// TwinCAT 3 PLC project RobotMainTask
// ProgramVersion: 3.1.4022.3
// libraries:
//   SysMem, * (System)
//   Tc2_MC2, * (Beckhoff Automation GmbH)
//   Tc2_SerialCom, * (Beckhoff Automation GmbH)
//   Tc2_Standard, * (Beckhoff Automation GmbH)
//   Tc2_System, * (Beckhoff Automation GmbH)
//   Tc2_TcpIp, * (Beckhoff Automation GmbH)
//   Tc3_Module, * (Beckhoff Automation GmbH)
// project tree:
//   / CommTask.TcTTO, MainTask.TcTTO
//   DUTs/ E_ExeCmd.TcDUT, E_MotorStatus.TcDUT, ST_AxisOut.TcDUT, ST_MoveObj.TcDUT, ST_PLCGroupSetAxis.TcDUT, ST_PLCSetAxis.TcDUT
//   GVLs/ GVL.TcGVL
//   POUs/ Comm.TcPOU, MAIN.TcPOU
//   POUs/Fuctions/ FB_ReadAxisStatus.TcPOU, FB_Robot.TcPOU, FB_SetAxisMotion.TcPOU, FB_RecvDataQue.TcPOU, FB_SendDataQue.TcPOU, FB_ServerWait.TcPOU
// real-time tasks:
//   TASK MainTask: cycle T#10ms, priority 8, ADS port 351
//   TASK CommTask: cycle T#20ms, priority 12, ADS port 352
// motion (NC):
//   TASK NC-Task 1 SAF: cycle T#2ms, priority 4, ADS port 501
//   TASK NC-Task 1 SVB: cycle T#10ms, priority 10, ADS port 511
//   AXIS Axis 1 (id 1)
//     OtherSettings: AllowMotionCmdToSlave=true
//     encoder EncType=19
//       EncPara: Offset=1210, MaxCount=#xffffffff
//     drive DrvType=16
//       DrvPara: MaxCount=#xffffffff, DriveControlDWord=#x00020000
//         Analog: ScaleFactorActTorque=0.1
//         TimeComp: TaskDelayCycles=1
//     controller CtrType=1
//       CtrPara: PriorControlFactor=1
//         Observer: BandWidth=20
//   AXIS Axis 2 (id 2)
//     OtherSettings: AllowMotionCmdToSlave=true
//     encoder EncType=19
//       EncPara: ScaleFactorDenominator=51.095748, Offset=1163.3371, Inverse=true, MaxCount=#xffffffff
//     drive DrvType=16
//       DrvPara: Inverse=true, MaxCount=#xffffffff, DriveControlDWord=#x00020000
//         Analog: ScaleFactorActTorque=0.1
//         TimeComp: TaskDelayCycles=1
//     controller CtrType=1
//       CtrPara: PriorControlFactor=1
//         Observer: BandWidth=20
//   AXIS Axis 3 (id 3)
//     OtherSettings: AllowMotionCmdToSlave=true
//     encoder EncType=19
//       EncPara: ScaleFactorDenominator=51.095748, Offset=318.369, Inverse=true, MaxCount=#xffffffff
//     drive DrvType=16
//       DrvPara: Inverse=true, MaxCount=#xffffffff, DriveControlDWord=#x00020000
//         Analog: ScaleFactorActTorque=0.1
//         TimeComp: TaskDelayCycles=1
//     controller CtrType=1
//       CtrPara: PriorControlFactor=1
//         Observer: BandWidth=20
//   AXIS Axis 4 (id 4)
//     OtherSettings: AllowMotionCmdToSlave=true
//     encoder EncType=19
//       EncPara: ScaleFactorDenominator=11.75751305, Offset=107.3187, Inverse=true, MaxCount=#xffffffff
//     drive DrvType=16
//       DrvPara: Inverse=true, MaxCount=#xffffffff, DriveControlDWord=#x00020000
//         Analog: ScaleFactorActTorque=0.1
//         TimeComp: TaskDelayCycles=1
//     controller CtrType=1
//       CtrPara: PriorControlFactor=1
//         Observer: BandWidth=20
//   AXIS Axis 5 (id 5)
//     OtherSettings: AllowMotionCmdToSlave=true
//     encoder EncType=19
//       EncPara: ScaleFactorDenominator=141.4214, Offset=4.8786, MaxCount=#xffffffff
//     drive DrvType=16
//       DrvPara: MaxCount=#xffffffff, DriveControlDWord=#x00020000
//         Analog: ScaleFactorActTorque=0.1
//         TimeComp: TaskDelayCycles=1
//     controller CtrType=1
//       CtrPara: PriorControlFactor=1
//         Observer: BandWidth=20
//   AXIS Axis 6 (id 6)
//     OtherSettings: AllowMotionCmdToSlave=true
//     encoder EncType=19
//       EncPara: ScaleFactorDenominator=5.22698, MaxCount=#xffffffff
//     drive DrvType=16
//       DrvPara: MaxCount=#xffffffff, DriveControlDWord=#x00020000
//         Analog: ScaleFactorActTorque=0.1
//         TimeComp: TaskDelayCycles=1
//     controller CtrType=1
//       CtrPara: PriorControlFactor=1
//         Observer: BandWidth=20
//   AXIS Axis 7 (id 7)
//     OtherSettings: AllowMotionCmdToSlave=true
//     encoder EncType=19
//       EncPara: ScaleFactorDenominator=5.25493, Offset=5, Inverse=true, MaxCount=#xffffffff
//     drive DrvType=16
//       DrvPara: Inverse=true, MaxCount=#xffffffff, DriveControlDWord=#x00020000
//         Analog: ScaleFactorActTorque=0.1
//         TimeComp: TaskDelayCycles=1
//     controller CtrType=1
//       CtrPara: PriorControlFactor=1
//         Observer: BandWidth=20
// I/O:
//   DEVICE Device 3 (EtherCAT), AmsNetId 192.168.1.240.4.1
//     Drive 1 (Elmo Drive) [Gold EtherCAT GCON Drive Rev:0x00010420]
//     Drive 2 (Elmo Drive) [Gold EtherCAT GCON Drive Rev:0x00010420]
//     Drive 3 (Elmo Drive) [Gold EtherCAT GCON Drive Rev:0x00010420]
//     Drive 4 (Elmo Drive) [Gold EtherCAT GCON Drive Rev:0x00010420]
//     Drive 5 (Elmo Drive) [Gold EtherCAT GCON Drive Rev:0x00010420]
//     Drive 6 (Elmo Drive) [Gold EtherCAT GCON Drive Rev:0x00010420]
//     Drive 7 (Elmo Drive) [Gold EtherCAT GCON Drive Rev:0x00010420]
//   DEVICE Device 2 (COM Port)
// variable links:
//   NC-Task 1 SAF/Axes/Axis 1 <-> Device 3 (EtherCAT)/Drive 1 (Elmo Drive)
//     Drive/Inputs/In/nDcOutputTime <-> InfoData/DcOutputShift
//     Drive/Inputs/In/nState1 <-> Inputs/Status word
//     Drive/Inputs/In/nState2 <-> Inputs/Status word @bit 8
//     Drive/Inputs/In/nState4 @bit 1 <-> WcState/InputToggle
//     Drive/Inputs/In/nState4 <-> WcState/WcState
//     Drive/Outputs/Out/nCtrl1 <-> Outputs/Control word
//     Drive/Outputs/Out/nCtrl2 <-> Outputs/Control word @bit 8
//     Drive/Outputs/Out/nDataOut1 <-> Outputs/Target Position
//     Enc/Inputs/In/nDataIn1 <-> Inputs/Position actual value
//     Enc/Inputs/In/nDcInputTime <-> InfoData/DcInputShift
//     Enc/Inputs/In/nState4 @bit 1 <-> WcState/InputToggle
//     Enc/Inputs/In/nState4 <-> WcState/WcState
//   NC-Task 1 SAF/Axes/Axis 2 <-> Device 3 (EtherCAT)/Drive 2 (Elmo Drive)
//     Drive/Inputs/In/nDcOutputTime <-> InfoData/DcOutputShift
//     Drive/Inputs/In/nState1 <-> Inputs/Status word
//     Drive/Inputs/In/nState2 <-> Inputs/Status word @bit 8
//     Drive/Inputs/In/nState4 @bit 1 <-> WcState/InputToggle
//     Drive/Inputs/In/nState4 <-> WcState/WcState
//     Drive/Outputs/Out/nCtrl1 <-> Outputs/Control word
//     Drive/Outputs/Out/nCtrl2 <-> Outputs/Control word @bit 8
//     Drive/Outputs/Out/nDataOut1 <-> Outputs/Target Position
//     Enc/Inputs/In/nDataIn1 <-> Inputs/Position actual value
//     Enc/Inputs/In/nDcInputTime <-> InfoData/DcInputShift
//     Enc/Inputs/In/nState4 @bit 1 <-> WcState/InputToggle
//     Enc/Inputs/In/nState4 <-> WcState/WcState
//   NC-Task 1 SAF/Axes/Axis 3 <-> Device 3 (EtherCAT)/Drive 3 (Elmo Drive)
//     Drive/Inputs/In/nDcOutputTime <-> InfoData/DcOutputShift
//     Drive/Inputs/In/nState1 <-> Inputs/Status word
//     Drive/Inputs/In/nState2 <-> Inputs/Status word @bit 8
//     Drive/Inputs/In/nState4 @bit 1 <-> WcState/InputToggle
//     Drive/Inputs/In/nState4 <-> WcState/WcState
//     Drive/Outputs/Out/nCtrl1 <-> Outputs/Control word
//     Drive/Outputs/Out/nCtrl2 <-> Outputs/Control word @bit 8
//     Drive/Outputs/Out/nDataOut1 <-> Outputs/Target Position
//     Enc/Inputs/In/nDataIn1 <-> Inputs/Position actual value
//     Enc/Inputs/In/nDcInputTime <-> InfoData/DcInputShift
//     Enc/Inputs/In/nState4 @bit 1 <-> WcState/InputToggle
//     Enc/Inputs/In/nState4 <-> WcState/WcState
//   NC-Task 1 SAF/Axes/Axis 4 <-> Device 3 (EtherCAT)/Drive 4 (Elmo Drive)
//     Drive/Inputs/In/nDcOutputTime <-> InfoData/DcOutputShift
//     Drive/Inputs/In/nState1 <-> Inputs/Status word
//     Drive/Inputs/In/nState2 <-> Inputs/Status word @bit 8
//     Drive/Inputs/In/nState4 @bit 1 <-> WcState/InputToggle
//     Drive/Inputs/In/nState4 <-> WcState/WcState
//     Drive/Outputs/Out/nCtrl1 <-> Outputs/Control word
//     Drive/Outputs/Out/nCtrl2 <-> Outputs/Control word @bit 8
//     Drive/Outputs/Out/nDataOut1 <-> Outputs/Target Position
//     Enc/Inputs/In/nDataIn1 <-> Inputs/Position actual value
//     Enc/Inputs/In/nDcInputTime <-> InfoData/DcInputShift
//     Enc/Inputs/In/nState4 @bit 1 <-> WcState/InputToggle
//     Enc/Inputs/In/nState4 <-> WcState/WcState
//   NC-Task 1 SAF/Axes/Axis 5 <-> Device 3 (EtherCAT)/Drive 5 (Elmo Drive)
//     Drive/Inputs/In/nDcOutputTime <-> InfoData/DcOutputShift
//     Drive/Inputs/In/nState1 <-> Inputs/Status word
//     Drive/Inputs/In/nState2 <-> Inputs/Status word @bit 8
//     Drive/Inputs/In/nState4 @bit 1 <-> WcState/InputToggle
//     Drive/Inputs/In/nState4 <-> WcState/WcState
//     Drive/Outputs/Out/nCtrl1 <-> Outputs/Control word
//     Drive/Outputs/Out/nCtrl2 <-> Outputs/Control word @bit 8
//     Drive/Outputs/Out/nDataOut1 <-> Outputs/Target Position
//     Enc/Inputs/In/nDataIn1 <-> Inputs/Position actual value
//     Enc/Inputs/In/nDcInputTime <-> InfoData/DcInputShift
//     Enc/Inputs/In/nState4 @bit 1 <-> WcState/InputToggle
//     Enc/Inputs/In/nState4 <-> WcState/WcState
//   NC-Task 1 SAF/Axes/Axis 6 <-> Device 3 (EtherCAT)/Drive 6 (Elmo Drive)
//     Drive/Inputs/In/nDataIn3[0] <-> Inputs_1/Torque actual value
//     Drive/Inputs/In/nDcOutputTime <-> InfoData/DcOutputShift
//     Drive/Inputs/In/nState1 <-> Inputs/Status word
//     Drive/Inputs/In/nState2 <-> Inputs/Status word @bit 8
//     Drive/Inputs/In/nState4 @bit 1 <-> WcState/InputToggle
//     Drive/Inputs/In/nState4 <-> WcState/WcState
//     Drive/Outputs/Out/nCtrl1 <-> Outputs/Control word
//     Drive/Outputs/Out/nCtrl2 <-> Outputs/Control word @bit 8
//     Drive/Outputs/Out/nDataOut1 <-> Outputs/Target Position
//     Enc/Inputs/In/nDataIn1 <-> Inputs/Position actual value
//     Enc/Inputs/In/nDcInputTime <-> InfoData/DcInputShift
//     Enc/Inputs/In/nState4 @bit 1 <-> WcState/InputToggle
//     Enc/Inputs/In/nState4 <-> WcState/WcState
//   NC-Task 1 SAF/Axes/Axis 7 <-> Device 3 (EtherCAT)/Drive 7 (Elmo Drive)
//     Drive/Inputs/In/nDcOutputTime <-> InfoData/DcOutputShift
//     Drive/Inputs/In/nState1 <-> Inputs/Status word
//     Drive/Inputs/In/nState2 <-> Inputs/Status word @bit 8
//     Drive/Inputs/In/nState4 @bit 1 <-> WcState/InputToggle
//     Drive/Inputs/In/nState4 <-> WcState/WcState
//     Drive/Outputs/Out/nCtrl1 <-> Outputs/Control word
//     Drive/Outputs/Out/nCtrl2 <-> Outputs/Control word @bit 8
//     Drive/Outputs/Out/nDataOut1 <-> Outputs/Target Position
//     Enc/Inputs/In/nDataIn1 <-> Inputs/Position actual value
//     Enc/Inputs/In/nDcInputTime <-> InfoData/DcInputShift
//     Enc/Inputs/In/nState4 @bit 1 <-> WcState/InputToggle
//     Enc/Inputs/In/nState4 <-> WcState/WcState
//   RobotMainTask/RobotMainTask Instance <-> Device 3 (EtherCAT)/Drive 6 (Elmo Drive)
//     CommTask Inputs/GVL.axisTorque <-> Inputs_1/Torque actual value
//   RobotMainTask/RobotMainTask Instance <-> NC-Task 1 SAF/Axes/Axis 1
//     MainTask Inputs/GVL.TestMotor[0].NcToPlc <-> Outputs/ToPlc
//     MainTask Outputs/GVL.TestMotor[0].PlcToNc <-> Inputs/FromPlc
//   RobotMainTask/RobotMainTask Instance <-> NC-Task 1 SAF/Axes/Axis 2
//     MainTask Inputs/GVL.TestMotor[1].NcToPlc <-> Outputs/ToPlc
//     MainTask Outputs/GVL.TestMotor[1].PlcToNc <-> Inputs/FromPlc
//   RobotMainTask/RobotMainTask Instance <-> NC-Task 1 SAF/Axes/Axis 3
//     MainTask Inputs/GVL.TestMotor[2].NcToPlc <-> Outputs/ToPlc
//     MainTask Outputs/GVL.TestMotor[2].PlcToNc <-> Inputs/FromPlc
//   RobotMainTask/RobotMainTask Instance <-> NC-Task 1 SAF/Axes/Axis 4
//     MainTask Inputs/GVL.TestMotor[3].NcToPlc <-> Outputs/ToPlc
//     MainTask Outputs/GVL.TestMotor[3].PlcToNc <-> Inputs/FromPlc
//   RobotMainTask/RobotMainTask Instance <-> NC-Task 1 SAF/Axes/Axis 5
//     MainTask Inputs/GVL.TestMotor[4].NcToPlc <-> Outputs/ToPlc
//     MainTask Outputs/GVL.TestMotor[4].PlcToNc <-> Inputs/FromPlc
//   RobotMainTask/RobotMainTask Instance <-> NC-Task 1 SAF/Axes/Axis 6
//     MainTask Inputs/GVL.TestMotor[5].NcToPlc <-> Outputs/ToPlc
//     MainTask Outputs/GVL.TestMotor[5].PlcToNc <-> Inputs/FromPlc
//   RobotMainTask/RobotMainTask Instance <-> NC-Task 1 SAF/Axes/Axis 7
//     MainTask Inputs/GVL.TestMotor[6].NcToPlc <-> Outputs/ToPlc
//     MainTask Outputs/GVL.TestMotor[6].PlcToNc <-> Inputs/FromPlc

CONFIGURATION RobotMainTask
    RESOURCE PLC ON TwinCAT3
        TASK CommTask(INTERVAL := T#20ms, PRIORITY := 12);
        TASK MainTask(INTERVAL := T#10ms, PRIORITY := 8);
        PROGRAM Comm WITH CommTask : Comm;
        PROGRAM MAIN WITH MainTask : MAIN;
    END_RESOURCE
END_CONFIGURATION

// ---- DUTs/E_ExeCmd.TcDUT
{attribute 'qualified_only'}
{attribute 'strict'}
TYPE E_ExeCmd :
(
		E_PowerOff,
		E_PowerOn,    //E_Enable
		E_MoveAbs,
		E_MoveConAbs,
		E_MoveRelative,
		E_MoveVelocity,
		E_Halt,
		E_Stop,
		E_Reset,
		E_Home
);
END_TYPE

// ---- DUTs/E_MotorStatus.TcDUT
{attribute 'qualified_only'}
{attribute 'strict'}
TYPE E_MotorStatus :
(
	MOTORSTATUS_DISABLED,       	//*****NEW	if the MC_Power.Enable is FALSE that motor will be disable, from any MOTORSTATUS
	MOTORSTATUS_Standstill,		//is the enable status, can response any Cmd
	MOTORSTATUS_ERRORSTOP,		//NEW
	MOTORSTATUS_HOMING,			//NEW
	MOTORSTATUS_STOPPING,		//NEW
	MOTORSTATUS_DISCRETEMOTION,		//NEW
	MOTORSTATUS_CONTINUOUSMOTION,	//NEW
	MOTORSTATUS_SYNMOTION		//Advance
);
END_TYPE

// ---- DUTs/ST_AxisOut.TcDUT
TYPE ST_AxisOut :
STRUCT


	eStatus   : E_MotorStatus;
	
	Response 	: STRING;
	ENABLE     : BOOL;
	ServoDone  : BOOL;
	ServoBusy  : BOOL;
	ServoError : BOOL;
	ServoErrorID : UDINT;	
//get these variable from the READSTATUS().NcToPlc;	
//	ErrorCode:UDINT;//NC轴错误代码
//	AxisState:UDINT;//NC轴状态
//	HomingState:UDINT;//NC轴回原位状态
//	AxisId:UDINT;//NC轴的编码
	ActPos:LREAL;//NC轴的实际位置
	ActVelo:LREAL;//NC轴的实际速度
	ActAcc:LREAL;//NC轴的实际加速度
	ActTorque:LREAL;//NC轴的实际转矩
	SetPos:LREAL;//NC轴的设定位置
	SetVelo:LREAL;//NC轴的设定速度
	SetAcc:LREAL;//NC轴的设定加速度
	SetTorque:LREAL;//NC轴的设定转矩
//	TargetPos:LREAL;//NC轴的目标位置
	PosDiff:LREAL;//位置误差	

END_STRUCT
END_TYPE

// ---- DUTs/ST_MoveObj.TcDUT
TYPE ST_MoveObj :
STRUCT
	
	Dir			: INT;	
	Position 		: LREAL;
	Distance 		: LREAL;
	Velocity 		: LREAL;
	EndVelocity 	: LREAL;
	Torque		: LREAL;

END_STRUCT
END_TYPE

// ---- DUTs/ST_PLCGroupSetAxis.TcDUT
TYPE ST_PLCGroupSetAxis :
STRUCT
	
	st_EachSetAxis : ARRAY [0..19] OF ST_PLCSetAxis;

END_STRUCT
END_TYPE

// ---- DUTs/ST_PLCSetAxis.TcDUT
TYPE ST_PLCSetAxis :
STRUCT
	
	Num  				: UINT;

	E_ExecuteCmd		: E_ExeCmd;
	ST_MoveObject		: ST_MoveObj;
		
END_STRUCT
END_TYPE

// ---- GVLs/GVL.TcGVL

{attribute 'qualified_only'}
VAR_GLOBAL
END_VAR
VAR_GLOBAL CONSTANT
	Reconnect_time 	: TIME := T#1S;
	ListenTime		: TIME := T#1S;
	AcceptTime		: TIME := T#1S;
	RecvTime 		: TIME := T#1S;	
	MaxDataLen		: UDINT := 3500;
	QueLen			: USINT := 4;
END_VAR
VAR_GLOBAL
	InitPar 		: st_InitParameter;
	// put new to tail and get data from heand  circularly
	fbRecvDataQue   : FB_RecvDataQue;
	fbSendDataQue 	: FB_SendDataQue;
	
	//NEW
	TestMotor : ARRAY [0..19] OF AXIS_REF;
END_VAR

// ---- POUs/Comm.TcPOU
PROGRAM Comm
VAR
	fbWaitConnect 	: FB_ServerWait;
	fbRecv			: FB_SocketReceive 	:= (sSrvNetId := '');
	fbSend			: FB_SocketSend 	:= (sSrvNetId := '');
	fbClose			: FB_SocketClose 	:= (sSrvNetID := '');	
	fbCloseAll		: FB_SocketCloseAll := (sSrvNetID := '');
	
	hSocket 		: T_HSOCKET;
	RecvLen 		: UDINT := 0;
	SendLen			: UDINT	:= 0;

	bNewRecv 		: BOOL;	
	bNewSend 		: BOOL;	
	bConnect 		: BOOL;
	nErrID 			: UDINT;
	step 			: UDINT;

	RecvBuff 		: ARRAY[1..GVL.MaxDataLen] OF BYTE;
	//SendBuff 		: ARRAY[1..GVL.DataLen] OF BYTE;
	SendBuff 		: ARRAY[1..GVL.MaxDataLen] OF BYTE;	
	DataRecv 		: ARRAY[1..GVL.MaxDataLen] OF BYTE;
	DataSend		: ARRAY[1..GVL.MaxDataLen] OF BYTE;
END_VAR

VAR(*For Test*)
	GetTime			: GETCPUACCOUNT;
	time_start		: UDINT;
	time_end 		: UDINT;
	time_cost 		: REAL;
END_VAR

CASE step OF
	0:(*prepare*)
		bConnect := FALSE;
		fbCloseAll(bExecute:= FALSE);
		fbCloseAll(bExecute:= TRUE);
		step := 1;
	1:(*Preparing*)
		fbCloseAll(bExecute:= FALSE);
		IF NOT fbCloseALL.bBusy THEN
			IF NOT fbCloseALL.bError THEN
				step := 5;
			ELSE 
				nErrID := fbCloseALL.nErrId;
				step := 0;
			END_IF
		END_IF
	5:(*wait for connect*)
		bConnect := FALSE;
		fbWaitConnect(bEnable := TRUE);
		nErrID := fbWaitConnect.nErrID;
		IF NOT fbWaitConnect.bBusy THEN
			IF NOT fbWaitConnect.bError THEN
				hSocket := fbWaitConnect.hSocket;
				step := 9;			
			ELSE
				nErrID := fbWaitConnect.nErrID;
			END_IF
		END_IF
		
	9:(*prepare to recieve data*)
		IF(GVL.InitPar.RecvSize <> 0) THEN
			fbRecv(bExecute := FALSE);
			bNewRecv := TRUE;
			bConnect := TRUE;
			RecvLen := GVL.InitPar.RecvSize;
			SendLen := GVL.InitPar.SendSize;
			step := 10;
			GVL.fbRecvDataQue.Reset();//Init recieve data queue
			GVL.fbSendDataQue.Reset();
		END_IF
		
		
	10:(*Receive and send phase I*)
		//*Start to recieve data
		fbRecv(hSocket := hSocket, cbLen := RecvLen, pDest := ADR(RecvBuff), bExecute := TRUE, tTimeout := GVL.RecvTime);
		//*prepare data to send
		fbSend(bExecute := FALSE);
		//Get SendData
		IF NOT fbSend.bBusy THEN
			IF NOT fbSend.bError THEN
				GVL.fbSendDataQue.GetFromQue(ADR(DataSend));
				step := 15;
			ELSE
				nErrID := fbSend.nErrId;
				step := 100;
			END_IF
		END_IF		
		step := 15;
	15: (*Receive and send phase II*)
		//deal with recieve data
		fbRecv(bExecute := FALSE);
		IF NOT fbRecv.bBusy THEN
			IF NOT fbRecv.bError THEN
				ACT_RecvData();
				IF bNewRecv THEN (*put databuff into recieve queque*)
					GVL.fbRecvDataQue.PutToQue(ADR(DataRecv));	
					memset(ADR(DataRecv),0, GVL.InitPar.RecvSize);		
				END_IF
				step := 10;			
			ELSE
				nErrID := fbRecv.nErrId;
				step := 100;	
			END_IF
		END_IF
		//SendData
		GVL.fbSendDataQue.GetFromQue(ADR(DataSend));
		
		IF GVL.fbSendDataQue.bGetData THEN
			fbSend(hSocket := hSocket,cbLen :=SendLen, pSrc := ADR(DataSend),bExecute := TRUE,tTimeout := gvl.RecvTime);
		END_IF
	100:(*deal with error*)
		bConnect := FALSE;
		fbClose(bExecute := FALSE);
		fbClose(hSocket := hSocket, bExecute := TRUE);
		step := 102;
	102: 
		bConnect := FALSE;
		fbClose(bExecute := FALSE);
		IF NOT fbClose.bBusy THEN
			IF NOT fbClose.bError THEN
				step:= 5;
			ELSE 
				step := 0;
			END_IF
		END_IF			
END_CASE

ACTION ACT_PreSend:

END_ACTION

ACTION ACT_RecvData:
(*Recieve data, every group of data has length of Datalen*)
IF bNewRecv THEN
	IF fbRecv.nRecBytes < GVL.InitPar.RecvSize THEN
		bNewRecv := FALSE;
		memcpy(ADR(DataRecv),ADR(RecvBuff),fbRecv.nRecBytes);
		RecvLen := GVL.InitPar.RecvSize - fbRecv.nRecBytes;
	ELSE
		memcpy(ADR(DataRecv),ADR(RecvBuff),GVL.InitPar.RecvSize);
		bNewRecv := TRUE;
	END_IF
ELSE
	IF fbRecv.nRecBytes < RecvLen THEN
		memcpy(ADR(DataRecv)+ GVL.InitPar.RecvSize - RecvLen, ADR(RecvBuff),fbRecv.nRecBytes);
		RecvLen := RecvLen - fbRecv.nRecBytes;
	ELSE		
		memcpy(ADR(DataRecv)+ GVL.InitPar.RecvSize - RecvLen, ADR(RecvBuff),RecvLen);
		bNewRecv := TRUE;
		RecvLen :=GVL.InitPar.RecvSize;
	END_IF					
END_IF
END_ACTION

END_PROGRAM

// ---- POUs/Fuctions/FB_ServerWait.TcPOU
FUNCTION_BLOCK FB_ServerWait
(*Listioning and accecpt connect for remote*)
VAR_INPUT
	bEnable : BOOL;
	sLocalHost : STRING(15) := '192.168.1.245';//'192.168.1.245';'192.168.137.74'
	nLocalPort : UINT := 4999;

END_VAR
VAR_OUTPUT
	hSocket : T_HSOCKET;
	bBusy: BOOL;
	bError: BOOL;
	nErrID : UDINT;
END_VAR
VAR
	fblisten :FB_SocketListen := (sSrvNetID := '');	
	fbAccept : FB_SocketAccept;
	fbClose : FB_SocketClose;
	fbReconncetTon: TON:=(PT := GVL.Reconnect_time);
	fbAcceptTon: TON:=(PT := GVL.AcceptTime);
		
	hListener : T_HSOCKET;	
	
	bListening : BOOL;
	bAccepting : BOOL;
	
	step : UINT := 0;
	
END_VAR

CASE step OF
	0:(*Init*)
		IF bEnable THEN
			fbReconncetTon(IN := FALSE);
			fblisten(bExecute := FALSE);
			step := 10;
			bBusy:= TRUE;
			nErrID := 0;
			bError := FALSE;
		END_IF
	10:(*Start listenin*)
		fbReconncetTon(IN := TRUE, PT := GVL.Reconnect_time);
		IF fbReconncetTon.Q THEN
			fblisten(sLocalHost := sLocalHost,
			nLocalPort := nLocalPort,
			bExecute := TRUE,
			tTimeout := GVL.ListenTime);
			step := 15;	
		END_IF
						
	15:(*Listening*)
		fbListen(bExecute := FALSE);
		bListening := TRUE;
		IF NOT fbListen.bBusy THEN
			IF NOT fbListen.bError THEN
				hListener := fbListen.hListener; 
				
				step := 20;
				(*prepare for accept*)
				fbAcceptTon(IN:=FALSE);
				fbAccept(bExecute := FALSE);
			ELSE
				bError := TRUE;				
				nErrID := fbListen.nErrId;
				step := 100;
			END_IF
		END_IF
	20:(*start to accept*)	
		bListening := FALSE;
		fbAcceptTon(IN := TRUE,PT := GVL.AcceptTime);
		IF fbAcceptTon.Q THEN
			fbAcceptTon(IN :=FALSE);
			fbAccept(hListener := hListener, bExecute := TRUE);
			step := 25;
		END_IF
	25: (* Accepting*)
		fbAccept(bExecute := FALSE);
		bAccepting := TRUE;
		IF NOT fbAccept.bBusy THEN
			IF NOT fbAccept.bError THEN
				(*check if there is connection be accepted*)
				IF fbAccept.bAccepted THEN
					hSocket := fbAccept.hSocket;
					bBusy := FALSE;
					step := 40;
				ELSE
					step := 20;
				END_IF	
							
			ELSE
				bError := TRUE;
				nErrID := fbAccept.nErrId;
				step := 100;	
			END_IF
		END_IF
		
	40:(*wait for new connect*)
		bBusy := TRUE;
		step:= 20;
	100:(*deal with error*)
		step := 0;
		
		
END_CASE

END_FUNCTION_BLOCK

// ---- POUs/MAIN.TcPOU

 PROGRAM MAIN
VAR{varable needed}
	robot				: FB_Robot;
	fbReadAxisStatus 	: FB_ReadAxisStatus;
	fbMCMotion 			: ARRAY[0..19] OF FB_SetAxisMotion;
	
	MC_ActStatus		: st_AxisGroupRead; 		 //**OUT**give the data to thr Upper
	MC_SetCommd			: st_AxisGroupSet;			 //**IN** get the data from the Upper and set the Axis 
	CtlComd		: RecvBuff;		(*Commd to MC*)
	Status		: SendBuff;		(*MC_State*)
	
	
	ErrID		: UDINT := 0;	
	step		: INT := 0;
	{time cost of every cycle}
	CycleTime	: LREAL := 0;
	CycleTime_Max: LREAL := 0;	
END_VAR

VAR{varable FOR test}
	i :UDINT := 0;
	j :UDINT := 0;
	w :UDINT := 0;
	vel : LREAL;
	nCounter: BYTE := 0;
	nCounter1: BYTE := 0;
	GetTime:GETCPUACCOUNT;
	time_start: UDINT;
	time_end:UDINT;
	labelOld:DINT := 0;
	labelNew:DINT := 0;
	count: UDINT := 0;
	count11 : UDINT := 0;
	delay : TON;
	
	test : LREAL := 0;
	test1 : LREAL := 0;
END_VAR

CASE step OF
	0: {prepare varable before start robot}	
		step := 5;
	5:	{NC init before robot start}	
		GroupInitAxis(); 	
		step := 10;
	10:{Init robot}
		ErrID := robot.InitRobot(ADR(GVL.InitPar));
	 	IF (0 = ErrID )THEN
		 	step := 15;
		ELSE
			step := 0;
		END_IF
	15:
		GetTime(cpuAccountDW=>time_start);
	 	
		GVL.fbRecvDataQue.GetfromQue(ADR(CtlComd));
		GroupReadAxis();

		robot.RunRobot(pMC_Inputs := ADR(MC_ActStatus), pMC_Outputs := ADR(MC_SetCommd),
								pCtlComd	:= ADR(CtlComd) , pRobotStatus := ADR(Status));
														
		GroupSetAxis();
		GVL.fbSendDataQue.PutToQue(ADR(Status));
		
		GetTime(cpuAccountDW=>time_end);
		CycleTime := (time_end- time_start)/10000.0;
		CycleTime_Max:= MAX(CycleTime,CycleTime_Max);
	 	
	20: 
		robot.StopRobot();
		step:= 0;
END_CASE;

ACTION GroupInitAxis:
i := 0;
END_ACTION

ACTION GroupReadAxis:
FOR i:= 0 TO 7 DO //MC_ActStatus.Number
	fbReadAxisStatus(AxisRef := GVL.TestMotor[i], AxisStatus => MC_ActStatus.AxisGoup[i]);	
END_FOR
END_ACTION

ACTION GroupSetAxis:
FOR i:= 0 TO 7 DO //MC_ActStatus.Number
	fbMCMotion[i](axis := GVL.TestMotor[i], SetCmd := MC_SetCommd.AxisGroup[i], ActStatus := MC_ActStatus.AxisGoup[i]);
END_FOR
//fbMCMotion(axis := GVL.TestMotor[0], SetCmd := MC_SetCommd.AxisGroup[0], ActStatus := MC_ActStatus.AxisGoup[0]);
END_ACTION

END_PROGRAM

// ---- POUs/Fuctions/FB_Robot.TcPOU
FUNCTION_BLOCK FB_Robot
VAR_INPUT
END_VAR
VAR_OUTPUT
END_VAR
VAR
	{attribute 'TcInitSymbol'}
	oidInstance : OTCID;
	ipRobot : IRobot;
	hrInit : HRESULT;
END_VAR

METHOD FB_exit : BOOL
VAR_INPUT
	bInCopyCode : BOOL; // if TRUE, the exit method is called for exiting an instance that is copied afterwards (online change).
END_VAR
IF NOT bInCopyCode THEN
	FW_SafeRelease(ADR(ipRobot));
END_IF
END_METHOD

METHOD FB_init : BOOL
VAR_INPUT
	bInitRetains : BOOL; // if TRUE, the retain variables are initialized (warm start / cold start)
	bInCopyCode : BOOL;  // if TRUE, the instance afterwards gets moved into the copy code (online change)
END_VAR
IF NOT bInCopyCode THEN
	IF ipRobot = 0 THEN
		hrInit := FW_objMgr_GetObjectInstance(oid := oidInstance, iid:= TC_GLOBAL_IID_LIST.IID_IRobot,pipUnk := ADR(ipRobot)); 
	END_IF
END_IF
END_METHOD

{attribute 'c++_compatible'}
{attribute 'minimal_input_size' := '4'}
{attribute 'pack_mode' := '4'}
{warning 'add method implementation'}
METHOD InitRobot : UDINT
VAR_INPUT
	pInitPar	: POINTER TO st_InitParameter;
END_VAR
IF (ipRobot <> 0) THEN
	InitRobot := ipRobot.InitRobot(pInitPar);
END_IF
END_METHOD


{attribute 'c++_compatible'}
{attribute 'minimal_input_size' := '4'}
{attribute 'pack_mode' := '4'}


METHOD RunRobot : UDINT
VAR_INPUT
	pMC_Inputs	: POINTER TO st_AxisGroupRead;
	pMC_Outputs	: POINTER TO st_AxisGroupSet;
	pCtlComd	: POINTER TO Recvbuff;
	pRobotStatus	: POINTER TO Sendbuff;
END_VAR
IF (ipRobot <> 0) THEN
	RunRobot := ipRobot.RunRobot(pMC_Inputs, pMC_Outputs, pCtlComd, pRobotStatus);
END_IF
END_METHOD

{attribute 'c++_compatible'}
{attribute 'minimal_input_size' := '4'}
{attribute 'pack_mode' := '4'}
{warning 'add method implementation'}
METHOD StopRobot : HRESULT
IF (ipRobot <> 0) THEN
	StopRobot := ipRobot.StopRobot();
END_IF
END_METHOD

END_FUNCTION_BLOCK

// ---- POUs/Fuctions/FB_ReadAxisStatus.TcPOU
FUNCTION_BLOCK FB_ReadAxisStatus
VAR_IN_OUT

AxisRef : AXIS_REF;

END_VAR

VAR_OUTPUT

AxisStatus : st_ReadAxis;

END_VAR
VAR	
END_VAR

AxisRef.ReadStatus();  
AxisStatus.Position			:= AxisRef.NcToPlc.ActPos;
AxisStatus.Velocity			:= AxisRef.NcToPlc.ActVelo;
AxisStatus.Acceleration		:= AxisRef.NcToPlc.ActAcc;
AxisStatus.Torque		    := AxisRef.NcToPlc.ActTorque;
//AxisStatus.Current			:= AxisRef.NcToPlc.ActTorque;
AxisStatus.ErrorID			:= AxisRef.NcToPlc.ErrorCode;

IF AxisRef.Status.ErrorStop THEN
	AxisStatus.eState := eAxis_ERRORSTOP;
ELSIF AxisRef.Status.Disabled THEN
	AxisStatus.eState := eAxis_DISABLED;
ELSIF AxisRef.Status.StandStill THEN
	AxisStatus.eState := eAxis_STANDSTILL;
ELSIF AxisRef.Status.Homing THEN
	AxisStatus.eState := eAxis_HOMING;
ELSIF AxisRef.Status.Stopping THEN
	AxisStatus.eState := eAxis_STOPPING;
ELSIF AxisRef.Status.DiscreteMotion THEN
	AxisStatus.eState := eAxis_DISCRETEMOTION;
ELSIF AxisRef.Status.ContinuousMotion THEN
	AxisStatus.eState := eAxis_CONTINOUSMOTION;
ELSIF AxisRef.Status.SynchronizedMotion THEN
	AxisStatus.eState := eAxis_SYNCHRONIZEDMOTION;
ELSE
	AxisStatus.eState := eAxis_UNDEFINED;
END_IF

END_FUNCTION_BLOCK

// ---- POUs/Fuctions/FB_SetAxisMotion.TcPOU
FUNCTION_BLOCK FB_SetAxisMotion
VAR_IN_OUT
		axis : AXIS_REF;   			// the input axis
END_VAR
VAR_INPUT
	SetCmd : st_SetAxis;	
	ActStatus: st_ReadAxis;
END_VAR
VAR		
	fbMC_Stop:			MC_Stop;		
	fbMC_Home:			MC_Home;		
	fbMC_Halt:			MC_Halt;
	fbMC_Power:			MC_Power;
	fbMC_Reset:			MC_Reset;
	fbMC_MovVel:		MC_MoveVelocity;
	fbMC_MovAbs:		MC_MoveAbsolute;
	fbMC_MovConAbs:		MC_MoveContinuousAbsolute;//定义一个绝对运动功能块
	fbMC_MovRelative:	MC_MoveRelative;	

	eDir				:mc_direction;
	
	bWarning			:BOOL := FALSE;
	
	bHalt				:BOOL := FALSE;
	

END_VAR

CASE ActStatus.eState OF
	
	eAxis_ERRORSTOP:
		A_ErrorStop();	
	eAxis_DISABLED:
		A_Disable();	
	eAxis_STANDSTILL:
		A_Standstill();
	eAxis_HOMING:
		A_Homing();		
	eAxis_STOPPING:
		A_Stopping();	
	eAxis_DISCRETEMOTION:
		A_DiscreteMotion();		
	eAxis_CONTINOUSMOTION:
		A_ContinuousMotion();			
END_CASE
fbMC_Stop( Axis:= axis,Execute:= FALSE );
fbMC_Halt(Axis:=axis, Execute:= FALSE);
fbMC_Home( Axis:=axis, Execute:=FALSE);
fbMC_Reset(Axis:= axis, 	Execute:=FALSE);
fbMC_MovAbs(Axis:= axis, Execute:=FALSE);
fbMC_MovConAbs(Axis:= axis, Execute:=FALSE);
fbMC_MovRelative(Axis:= axis,  Execute:=FALSE);
fbMC_MovVel(Axis:= axis, Execute:=FALSE);

ACTION A_ContinuousMotion:
CASE SetCmd.eMC_Motion OF
	eMC_NONE:
		//fbMC_Halt(Axis:=axis, Execute:= TRUE);
	eMC_POWER:
		IF SetCmd.bEnable = TRUE THEN
			fbMC_Power(	Axis:= axis, Enable:= TRUE, Enable_Positive:= TRUE,
					Enable_Negative:= TRUE );
		ELSE
			fbMC_Power(	Axis:= axis, Enable:= FALSE);			
		END_IF	
		
	eMC_STOP:
		fbMC_Stop( Axis:= axis,Execute:= TRUE );
//		fbMC_Stop( Axis:= axis,Execute:= FALSE );
	
	eMC_HALT:
		fbMC_Halt(Axis:=axis, Execute:= TRUE);
//		fbMC_Halt(Axis:=axis, Execute:= FALSE);
		
	eMC_MOV_ABS:
		fbMC_MovAbs(Axis:= axis, Execute:=TRUE , 
					Position:=SetCmd.Position, 
					Velocity:=ABS(SetCmd.Velocity),
					BufferMode := MC_BlendingLow);
//		fbMC_MovAbs(Axis:= axis, Execute:=FALSE);
	
	eMC_MOV_CON_ABS:
		fbMC_MovConAbs(Axis:= axis, Execute:=TRUE, 
						Position:=SetCmd.Position ,Velocity:= ABS(SetCmd.Velocity),
						EndVelocity:= ABS(SetCmd.EndVelocity));
//		fbMC_MovConAbs(Axis:= axis, Execute:=FALSE);
	
	eMC_MOV_RELATIVE:
		fbMC_MovRelative(Axis:= axis,  Execute:=TRUE , 
			Distance:= SetCmd.Distance,  Velocity:= SetCmd.Velocity);
//		fbMC_MovRelative(Axis:= axis,  Execute:=FALSE);
	
	eMC_MOV_VEL:
		IF (SetCmd.Velocity >= 0) THEN
			eDir := MC_Positive_Direction;
		ELSE
			eDir := MC_Negative_Direction;
		END_IF
		fbMC_MovVel(Axis:= axis, Execute:=TRUE, 
					Velocity:=ABS(SetCmd.Velocity), Direction:=eDir);	
//		fbMC_MovVel(Axis:= axis, Execute:=FALSE);
		
ELSE
	bWarning := TRUE;
END_CASE
END_ACTION

ACTION A_Disable:
CASE SetCmd.eMC_Motion OF
	eMC_NONE:
	eMC_POWER:
		IF SetCmd.bEnable = TRUE THEN
			fbMC_Power(	Axis:= axis, Enable:= TRUE, Enable_Positive:= TRUE,
					Enable_Negative:= TRUE );
		ELSE
			fbMC_Power(	Axis:= axis, Enable:= FALSE);			
		END_IF
	eMC_Reset:
		fbMC_Reset(Axis:= axis, 	Execute:=TRUE);
//		fbMC_Reset(Axis:= axis, 	Execute:=FALSE);	
ELSE
	bWarning := TRUE;
END_CASE
END_ACTION

ACTION A_DiscreteMotion:
CASE SetCmd.eMC_Motion OF
	eMC_NONE:
		//fbMC_Halt(Axis:=axis, Execute:= TRUE);			
	eMC_POWER:
		IF SetCmd.bEnable = TRUE THEN
			fbMC_Power(	Axis:= axis, Enable:= TRUE, Enable_Positive:= TRUE,
					Enable_Negative:= TRUE );
		ELSE
			fbMC_Power(	Axis:= axis, Enable:= FALSE);			
		END_IF
	
	eMC_STOP:
		fbMC_Stop( Axis:= axis,Execute:= TRUE );
//		fbMC_Stop( Axis:= axis,Execute:= FALSE );
	
	eMC_HALT:
		fbMC_Halt(Axis:=axis, Execute:= TRUE);
//		fbMC_Halt(Axis:=axis, Execute:= FALSE);

	eMC_MOV_ABS:
		fbMC_MovAbs(Axis:= axis, Execute:=TRUE , 
					Position:=SetCmd.Position, 
					Velocity:=ABS(SetCmd.Velocity),
					BufferMode := MC_BlendingLow);
//		fbMC_MovAbs(Axis:= axis, Execute:=FALSE);
	
	eMC_MOV_CON_ABS:
		fbMC_MovConAbs(Axis:= axis, Execute:=TRUE, 
						Position:=SetCmd.Position ,Velocity:= ABS(SetCmd.Velocity),
						EndVelocity:= ABS(SetCmd.EndVelocity));
//		fbMC_MovConAbs(Axis:= axis, Execute:=FALSE);
	
	eMC_MOV_RELATIVE:
		fbMC_MovRelative(Axis:= axis,  Execute:=TRUE , 
			Distance:= SetCmd.Distance,  Velocity:= SetCmd.Velocity);
//		fbMC_MovRelative(Axis:= axis,  Execute:=FALSE);
	
	eMC_MOV_VEL:
		IF (SetCmd.Velocity >= 0) THEN
			eDir := MC_Positive_Direction;
		ELSE
			eDir := MC_Negative_Direction;
		END_IF
		fbMC_MovVel(Axis:= axis, Execute:=TRUE, 
					Velocity:=ABS(SetCmd.Velocity), Direction:=eDir);	
//		fbMC_MovVel(Axis:= axis, Execute:=FALSE);
		
ELSE
	bWarning := TRUE;
END_CASE
END_ACTION

ACTION A_ErrorStop:
CASE SetCmd.eMC_Motion OF
	eMC_NONE:
	eMC_RESET:	
		fbMC_Reset(Axis:= axis, 	Execute:=TRUE);		
//		fbMC_Reset(Axis:= axis, 	Execute:=FALSE);	
ELSE
	bWarning := TRUE;
END_CASE
END_ACTION

ACTION A_Homing:
CASE SetCmd.eMC_Motion OF
	eMC_NONE:	
	eMC_STOP:
		fbMC_Stop(Axis:=axis, 	Execute:=TRUE);
//		fbMC_Stop(Axis:=axis, 	Execute:=FALSE);
	eMC_POWER:
		IF SetCmd.bEnable = TRUE THEN
			fbMC_Power(	Axis:= axis, Enable:= TRUE, Enable_Positive:= TRUE,
					Enable_Negative:= TRUE );
		ELSE
			fbMC_Power(	Axis:= axis, Enable:= FALSE);			
		END_IF
ELSE
	bWarning := TRUE;		
END_CASE
END_ACTION

ACTION A_Standstill:
CASE SetCmd.eMC_Motion OF
	eMC_NONE:
	eMC_RESET:
		fbMC_Reset(Axis:= axis, 	Execute:=TRUE);

		bWarning := TRUE;	
	eMC_HOME:
		fbMC_Home( Axis:=axis, Execute:=TRUE ,
				   Position:=0 ,HomingMode:= );

	
	eMC_POWER:
		IF SetCmd.bEnable = TRUE THEN
			fbMC_Power(	Axis:= axis, Enable:= TRUE, Enable_Positive:= TRUE,
					Enable_Negative:= TRUE );
		ELSE
			fbMC_Power(	Axis:= axis, Enable:= FALSE);			
		END_IF	
		
	eMC_STOP:
		fbMC_Stop( Axis:= axis,Execute:= TRUE );

	
	eMC_HALT:
		fbMC_Halt(Axis:=axis, Execute:= TRUE);


	eMC_MOV_ABS:

		fbMC_MovAbs(Axis:= axis, Execute:=TRUE , 
					Position:= SetCmd.Position, 
					Velocity:= ABS(SetCmd.Velocity));

	
	eMC_MOV_CON_ABS:
		fbMC_MovConAbs(Axis:= axis, Execute:=TRUE, 
						Position:= SetCmd.Position ,Velocity:= ABS(SetCmd.Velocity),
						EndVelocity:= ABS(SetCmd.EndVelocity));

	
	eMC_MOV_RELATIVE:
		fbMC_MovRelative(Axis:= axis,  Execute:=TRUE , 
			Distance:= SetCmd.Distance,  Velocity:= ABS(SetCmd.Velocity));

	
	eMC_MOV_VEL:
		IF (SetCmd.Velocity >= 0) THEN
			eDir := MC_Positive_Direction;
		ELSE
			eDir := MC_Negative_Direction;
		END_IF
		fbMC_MovVel(Axis:= axis, Execute:=TRUE, 
					Velocity:=ABS(SetCmd.Velocity), Direction:=eDir);

ELSE
	bWarning := TRUE;	
END_CASE
END_ACTION

ACTION A_Stopping:
CASE SetCmd.eMC_Motion OF
	eMC_NONE:
	eMC_STOP:
		fbMC_Stop( Axis:= axis,Execute:= TRUE );
//		fbMC_Stop( Axis:= axis,Execute:= FALSE );		
	eMC_POWER:
		IF SetCmd.bEnable = TRUE THEN
			fbMC_Power(	Axis:= axis, Enable:= TRUE, Enable_Positive:= TRUE,
					Enable_Negative:= TRUE );
		ELSE
			fbMC_Power(	Axis:= axis, Enable:= FALSE);			
		END_IF
	
ELSE
	bWarning := TRUE;
END_CASE
END_ACTION

END_FUNCTION_BLOCK

// ---- POUs/Fuctions/FB_RecvDataQue.TcPOU
FUNCTION_BLOCK FB_RecvDataQue
VAR_INPUT
END_VAR
VAR_OUTPUT
END_VAR
VAR
	nQueHead			: USINT := 1;
	nQueTail			: USINT := 0;
	i					: USINT := 0;
	GetDataFailCNT		: UDINT := 0;
	PutDataFailCNT		: UDINT := 0;
END_VAR
VAR (*DATA ACCESS BY SERVAL TASK*)
	bRecvQueFill		: ARRAY[1..GVL.QueLen] OF BOOL;
	bRecvQueLock		: ARRAY[1..GVL.QueLen] OF BOOL;
	RecvQue				: ARRAY[1..GVL.QueLen, 1..GVL.MaxDataLen] OF BYTE;
END_VAR

METHOD GetfromQue : BOOL
VAR_INPUT
	DataBuff 		: POINTER TO ARRAY[1..GVL.MaxDataLen] OF BYTE;
END_VAR
IF TestAndSet(bRecvQueLock[nQueHead])THEN
	IF bRecvQueFill[nQueHead] THEN
		memcpy(DataBuff,ADR(RecvQue)+ (nQueHead-1)*GVL.MaxDataLen,GVL.MaxDataLen);
		bRecvQueLock[nQueHead]:= FALSE;	
		
		bRecvQueFill[nQueHead]:= FALSE;
		nQueHead := nQueHead + 1;
		GetDataFailCNT := 0;
		IF nQueHead > 4 THEN
			nQueHead := 1;
		END_IF
	ELSE
		memset(DataBuff,0,GVL.MaxDataLen);
		bRecvQueLock[nQueHead]:= FALSE;	
		GetDataFailCNT := GetDataFailCNT+1;			
	END_IF
	
ELSE
	//the que is emty, set buffer 0.
	memset(DataBuff,0,GVL.MaxDataLen);
	GetDataFailCNT := GetDataFailCNT+1;
END_IF
END_METHOD

METHOD PUBLIC PutToQue : BOOL
VAR_INPUT
	DataBuff 		: POINTER TO ARRAY[1..GVL.MaxDataLen] OF BYTE;
END_VAR
nQueTail := nQueTail + 1;
IF nQueTail > 4 THEN
	nQueTail := 1;
END_IF
IF TestAndSet(bRecvQueLock[nQueTail])THEN
	memcpy(ADR(RecvQue)+ (nQueTail-1)*GVL.MaxDataLen,DataBuff,GVL.MaxDataLen);
	bRecvQueLock[nQueTail]:= FALSE;	
	bRecvQueFill[nQueTail]:= TRUE;
	PutDataFailCNT := 0;
	
ELSE
	//abandan this data, this may cause unresbonse to some command (very very low possiblity)
	nQueTail := nQueTail - 1;
	IF nQueTail = 0 THEN
	nQueTail := 4;
	END_IF
	PutDataFailCNT := PutDataFailCNT+1;
END_IF
END_METHOD

METHOD Reset : BOOL
VAR_INPUT
END_VAR
FOR i := 1 TO GVL.QueLen DO
	IF TestAndSet(bRecvQueLock[i]) THEN
		bRecvQueFill[i] := FALSE;
		bRecvQueLock[i] := FALSE;
	END_IF
END_FOR
nQueHead := 1;
nQueTail := 0;
END_METHOD

END_FUNCTION_BLOCK

// ---- POUs/Fuctions/FB_SendDataQue.TcPOU
FUNCTION_BLOCK FB_SendDataQue
VAR

END_VAR
VAR (*DATA ACCESS BY SERVAL TASK*)
	bSendQueFill		: BOOL;
	bSendQueLock		: BOOL;
	SendQue				: ARRAY[1..GVL.MaxDataLen] OF BYTE;
	
	GetDataFailCNT		: UDINT := 0;
	PutDataFailCNT		: UDINT := 0;
END_VAR

VAR_OUTPUT
	bGetData			: BOOL;
END_VAR

METHOD GetFromQue : BOOL
VAR_INPUT
	DataBuff 		: POINTER TO ARRAY[1..GVL.MaxDataLen] OF BYTE;
END_VAR
IF TestAndSet(bSendQueLock)THEN
	IF bSendQueFill THEN
		memcpy(DataBuff,ADR(SendQue),GVL.MaxDataLen);	
		bSendQueFill:= FALSE;
		bGetData := TRUE;
		GetDataFailCNT := 0;
	ELSE 
		memcpy(DataBuff,0,SIZEOF(DataBuff));
		GetDataFailCNT := GetDataFailCNT+1;
		bGetData := FALSE;
	END_IF
	bSendQueLock:= FALSE;	
ELSE
	//the que is emty, set buffer 0.
	memset(DataBuff,0,SIZEOF(DataBuff));
	GetDataFailCNT := GetDataFailCNT+1;
	bGetData := FALSE;
END_IF
END_METHOD

METHOD PutToQue : BOOL
VAR_INPUT
	DataBuff 		: POINTER TO ARRAY[1..GVL.MaxDataLen] OF BYTE;
END_VAR
IF TestAndSet(bSendQueLock) THEN
	memcpy(ADR(SendQue),DataBuff,GVL.MaxDataLen);
	bSendQueFill:= TRUE;
	PutDataFailCNT := 0;
	
	bSendQueLock:= FALSE;
ELSE
	PutDataFailCNT := PutDataFailCNT + 1;
END_IF
END_METHOD

METHOD Reset : BOOL
VAR_INPUT
END_VAR
IF TestAndSet(bSendQueLock) THEN
	bSendQueFill:= FALSE;
	bGetData := FALSE;
	
	bSendQueLock:= FALSE;	
END_IF
END_METHOD

END_FUNCTION_BLOCK
